FUNCTION_BLOCK PAEDriveBase EXTENDS PAEControlModuleBase
VAR_INPUT
END_VAR
VAR_OUTPUT
END_VAR
VAR
	_MaintenanceSwitch : BOOL;
END_VAR

METHOD PUBLIC FB_postinit
VAR_INPUT
		root : IACVariobatch;
END_VAR
SUPER^.FB_postinit(root);
root.OnPropertyChangedBool(THIS^, 33, _MaintenanceSwitch);
END_METHOD

METHOD PUBLIC InvokeSetterBool
VAR_INPUT
	PropertyID : INT;
	PropertyValue : BOOL;
END_VAR
SUPER^.InvokeSetterBool(PropertyID, PropertyValue);
IF PropertyID = 33 THEN
	MaintenanceSwitch := PropertyValue;
END_IF
END_METHOD

{attribute 'monitoring' := 'call'}
//{attribute 'TcRpcEnable'}
PROPERTY PUBLIC MaintenanceSwitch : BOOL
GET // PUBLIC
MaintenanceSwitch := _MaintenanceSwitch;
END_GET
SET // PUBLIC
_MaintenanceSwitch := MaintenanceSwitch;
Root.OnPropertyChangedBool(THIS^, 33, _MaintenanceSwitch);
END_SET
END_PROPERTY

METHOD OnInitMemory
VAR_INPUT
		root : IACVariobatch;
END_VAR
RegisterProperty(root, 33, GCL.cSizeBYTE); //MaintenanceSwitch
SUPER^.OnInitMemory(root);
END_METHOD

END_FUNCTION_BLOCK

(* stored: Version 1.1.0.1, ProductVersion 3.1.4024.6
   POU PAEDriveBase: Id {45c98bb3-1009-4483-86de-a6e6e667dd40}, SpecialFunc None
   Method FB_postinit: Id {fdf6ebba-3975-4f15-9851-76b5aacc1960}
   Method InvokeSetterBool: Id {bbe82952-33a0-4f2f-b6ea-b83fbfec4041}
   Property MaintenanceSwitch: Id {1672a295-32d6-4a25-a713-7c703a14502b}
   Get Get: Id {69611494-b6cf-4dbf-a9da-2b76549f1408}
   Set Set: Id {18b00f6b-7c45-4f88-a7bb-a96b1901aba3}
   Method OnInitMemory: Id {565fa218-76f1-4c37-933d-cdd2d491010d} *)
